Staubli VAL3: onF6Event.pgx

program onF6Event(tool x_tTool, bool& x_bSave[])
  local string l_sMessage
  local string l_sName
  local num l_nSize
begin
  // look if the bButton is enable
  if bButton[5]
    //
    // DUPLICATE
    //
    call language:message(l_sMessage,126)
    call tcp:getName(l_sName,nIndexTool)
    popUpMsg(l_sMessage+l_sName)
    call tcp:new(x_tTool.trsf)
    call tcp:getSize(l_nSize)
    nIndexTool=l_nSize-1
    //    // refresh and modify the name
    call buildList()
    call refreshStatic()
    nIndex=0
    call editTool(x_tTool)
    logMsg("[KERNEL] INTERFACE:Insert new tool at index: "+toString("",l_nSize))
    x_bSave=true
  endIf
end
